(* IEC 61131-3 sources: stc/tests/fixtures/invalid_semantic, 2 files *)

(* ---- class_missing.st ---- *)
CLASS (* missing class name *)
	VAR PUBLIC
		p: INT := (* missing initializer value *) ;
	END_VAR
END_CLASS

FUNCTION SomeFuction
	RETURN 13 (* superfluous literal *) ;
END_FUNCTION

FUNCTION SomeOtherFunction
	a := 12;
	CLASS (* superfluous keyword *)
END_FUNCTION

(* ---- undeclared_variable.st ---- *)
(* Copyright (C) 2021-2026 Manuele Conti
   SPDX-License-Identifier: GPL-2.0-or-later
   Summary: Verifies diagnostics for references to undeclared variables. *)

FUNCTION bad : INT
VAR_INPUT
    input_value: INT;
END_VAR
    bad := input_value + missing_value;
END_FUNCTION
